# EPICS autosave request: ipApp/Db/USdigital_X3_settings.req
$(P)USdig_X3:$(S):A1.DESC
$(P)USdig_X3:$(S):A1.B
$(P)USdig_X3:$(S):A2.DESC
$(P)USdig_X3:$(S):A2.B
$(P)USdig_X3:$(S):A3.DESC
$(P)USdig_X3:$(S):A3.B
